// TIA Portal project "START_STOP_NODE_RED" (V19)

(* hardware
DEVICE "S7-1200 station_1"  S7-1200 Station
   slot 0: "Rack_0"  S7-1200 Rack  Rack  V1.0
   slot 1: "PLC_1"  CPU 1214C AC/DC/Rly  6ES7 214-1BE30-0XB0  V2.2
   slot 3: "AQ 1x12BIT_1"  AQ1 signal board  6ES7 232-4HA30-0XB0  V1.0
*)

// ===== PLC "PLC_1"  CPU 1214C AC/DC/Rly =====

VAR_GLOBAL   // PLC tag table "Default tag table"
   "Tag_1" AT %I0.0 : Bool;
   "BANDA" AT %Q0.0 : Bool;
   "SWITCH_ARRIBA" AT %I1.3 : Bool;
   "Tag_3" AT %Q0.2 : Bool;
   "Tag_4" AT %Q0.1 : Bool;
   "SWITCH_ABAJO" AT %I1.2 : Bool;
   "Tag_2" AT %IW64 : Int;
   "Tag_5" AT %MD2 : Real;
   "PORCENTAJE" AT %MW10 : Int;
   "Tag_6" AT %I0.1 : Bool;
END_VAR

DATA_BLOCK "DATOS"   // DB1
{ S7_Optimized_Access := 'FALSE' }
VERSION : 0.1
   VAR
      START : Bool;
      STOP : Bool;
   END_VAR
BEGIN
END_DATA_BLOCK

ORGANIZATION_BLOCK "Main"   // OB1, LAD, ProgramCycle
TITLE = "Main Program Sweep (Cycle)"
{ S7_Optimized_Access := 'TRUE' }
VERSION : 0.1
BEGIN

REGION Network 1
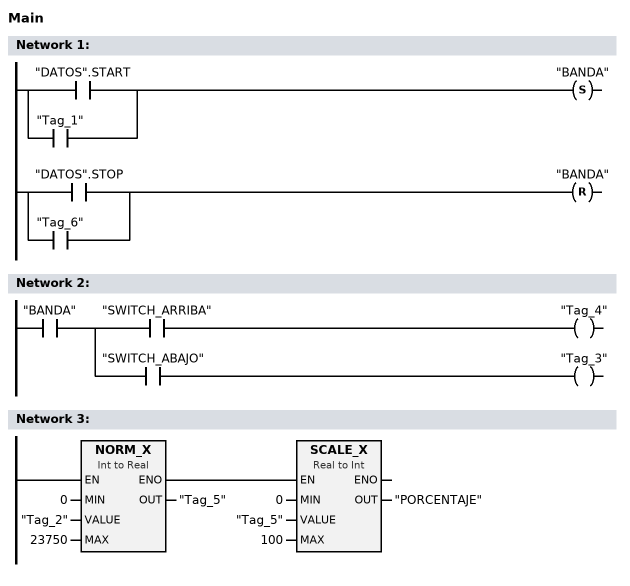
   RUNG wire#powerrail
      Contact( "DATOS".START )
      wire#w1
      S_Coil( "BANDA" )
   END_RUNG
   RUNG wire#powerrail
      Contact( "Tag_1" )
   END_RUNG wire#w1
   RUNG wire#powerrail
      Contact( "DATOS".STOP )
      wire#w2
      R_Coil( "BANDA" )
   END_RUNG
   RUNG wire#powerrail
      Contact( "Tag_6" )
   END_RUNG wire#w2
   // the same network as SCL:
   IF "DATOS".START OR "Tag_1" THEN "BANDA" := TRUE; END_IF;
   IF "DATOS".STOP OR "Tag_6" THEN "BANDA" := FALSE; END_IF;
END_REGION

REGION Network 2
   RUNG wire#powerrail
      Contact( "BANDA" )
      wire#w1
      Contact( "SWITCH_ARRIBA" )
      Coil( "Tag_4" )
   END_RUNG
   RUNG wire#w1
      Contact( "SWITCH_ABAJO" )
      Coil( "Tag_3" )
   END_RUNG
   // the same network as SCL:
   "Tag_4" := "BANDA" AND "SWITCH_ARRIBA";
   "Tag_3" := "BANDA" AND "SWITCH_ABAJO";
END_REGION

REGION Network 3
   RUNG wire#powerrail
      { S7_Templates := "[SrcType := Int, DestType := Real]"; S7_GenerateENO := "TRUE" } Normalize(min := 0, value := "Tag_2", max := 23750, out => "Tag_5")
      { S7_Templates := "[SrcType := Real, DestType := Int]"; S7_GenerateENO := "TRUE" } Scale(min := 0, value := "Tag_5", max := 100, out => "PORCENTAJE")
   END_RUNG
   // the same network as SCL:
   // ENO of a box is taken as its EN; it also drops when the box reports an error
   "Tag_5" := NORM_X(MIN := 0, VALUE := "Tag_2", MAX := 23750);
   "PORCENTAJE" := SCALE_X(MIN := 0, VALUE := "Tag_5", MAX := 100);
END_REGION
END_ORGANIZATION_BLOCK